/// Implicitly generated code : DO NOT EDIT!!!
/// Checks for division by 0, if divisor is 0, replace it with 1 and report error
{attribute 'check_div_int32' := ''}
{attribute 'no_check' := ''}
FUNCTION CheckDivDInt : DINT
VAR_INPUT
	divisor: DINT;
END_VAR

IF divisor = 0 THEN
	// replace divisor and report error if necessary
	CheckDivDInt := 1;
	GVL_Supervision.aCodeErr[eCodeError_divDInt] := TRUE;
ELSE
	CheckDivDInt := divisor;
END_IF;

END_FUNCTION

(* stored: Version 1.1.0.1, ProductVersion 3.1.4022.9
   POU CheckDivDInt: Id {5d5b7a29-d1ab-41a8-8a74-fc949448b71d}, SpecialFunc None *)
